Staubli VAL3: refreshDynamic.pgx

program refreshDynamic()
  local string l_sMessage
begin
//  // DO NOT CHANGE
  nRefresh=clock()
  use:bUseRefresh=false
//  //
//  // ADD HERE
//  //
end
